FUNCTION_BLOCK F_OR (* standard bitwise boolean OR function *)
  PACKAGE iec61131::arithmetic;
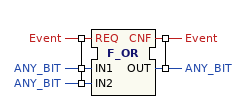
  EVENT_INPUT
    REQ WITH IN1, IN2; (* Service Request *)
  END_EVENT
  EVENT_OUTPUT
    CNF WITH OUT; (* Confirmation of Requested Service *)
  END_EVENT
  VAR_INPUT
    IN1 : ANY_BIT; (* Input *)
    IN2 : ANY_BIT; (* Input *)
  END_VAR
  VAR_OUTPUT
    OUT : ANY_BIT; (* Output *)
  END_VAR
  (* Service APPLICATION/RESOURCE: bitwise or *)
END_FUNCTION_BLOCK
